(*

short summary
=================
This interface provides assert statements for 32 bit ``DATE``  

.. <legal notes>

legal notes
=================
| SPDX-FileCopyrightText: © 2022 ekvip automation GmbH <info@ekvip.de>
| SPDX-License-Identifier: Apache-2.0
| For details check: Apache-2.0_

.. _Apache-2.0: https://www.apache.org/licenses/LICENSE-2.0

.. </legal notes>

methods
==================

*)

INTERFACE I64BitDateAssertions EXTENDS __SYSTEM.IQueryInterface

(*

short summary
=================
This assertion method checks if the current value is equal to the expected value

.. <legal notes>

legal notes
=================
| SPDX-FileCopyrightText: © 2022 ekvip automation GmbH <info@ekvip.de>
| SPDX-License-Identifier: Apache-2.0
| For details check: Apache-2.0_

.. _Apache-2.0: https://www.apache.org/licenses/LICENSE-2.0

.. </legal notes>

parameters
=================

*)

METHOD valueIsEqualTo
VAR_INPUT
	(* current value to check *)
	currentValue	:LDATE;
	(* expected value to compare *)
	expectedValue	:LDATE;
	(* message if the assertion is false *)
	message			:AssertMessage;
END_VAR
END_METHOD

(*

short summary
=================
This assertion method checks if the current value is greater than the less value

.. <legal notes>

legal notes
=================
| SPDX-FileCopyrightText: © 2022 ekvip automation GmbH <info@ekvip.de>
| SPDX-License-Identifier: Apache-2.0
| For details check: Apache-2.0_

.. _Apache-2.0: https://www.apache.org/licenses/LICENSE-2.0

.. </legal notes>

parameters
=================

*)

METHOD valueIsGreaterThan
VAR_INPUT
	(* current value to check *)
	currentValue	:LDATE;
	(* less than lower limit *)
	lessValue		:LDATE;
	(* message if the assertion is false *)
	message			:AssertMessage;
END_VAR
END_METHOD

(*

short summary
=================
This assertion method checks if the current value is inside a limit

.. attention:: 
	limits are included: ``valueIsInRangeOf(ldate#1970-01-01, ldate#1970-01-01, ldate#1970-01-01)``
	is a true assertion

.. <legal notes>

legal notes
=================
| SPDX-FileCopyrightText: © 2022 ekvip automation GmbH <info@ekvip.de>
| SPDX-License-Identifier: Apache-2.0
| For details check: Apache-2.0_

.. _Apache-2.0: https://www.apache.org/licenses/LICENSE-2.0

.. </legal notes>

parameters
=================

*)

METHOD valueIsInRangeOf
VAR_INPUT
	(* lower limit for the current value *)
	lowerLimit		:LDATE;
	(* current value to check *)
	currentValue	:LDATE;
	(* upper limit for the current value *)
	upperLimit		:LDATE;
	(* message if the assertion is false *)
	message			:AssertMessage;
END_VAR
END_METHOD

(*

short summary
=================
This assertion method checks if the current value is less than the greater value

.. <legal notes>

legal notes
=================
| SPDX-FileCopyrightText: © 2022 ekvip automation GmbH <info@ekvip.de>
| SPDX-License-Identifier: Apache-2.0
| For details check: Apache-2.0_

.. _Apache-2.0: https://www.apache.org/licenses/LICENSE-2.0

.. </legal notes>

parameters
=================

*)

METHOD valueIsLessThan
VAR_INPUT
	(* current value to check *)
	currentValue	:LDATE;
	(* greater than upper limit *)
	greaterValue	:LDATE;
	(* message if the assertion is false *)
	message			:AssertMessage;
END_VAR
END_METHOD

(*

short summary
=================
This assertion method checks if the current value is less than or equal to the maximum value

.. <legal notes>

legal notes
=================
| SPDX-FileCopyrightText: © 2022 ekvip automation GmbH <info@ekvip.de>
| SPDX-License-Identifier: Apache-2.0
| For details check: Apache-2.0_

.. _Apache-2.0: https://www.apache.org/licenses/LICENSE-2.0

.. </legal notes>

parameters
=================

*)

METHOD valueIsMax
VAR_INPUT
	(* current value to check *)
	currentValue	:LDATE;
	(* upper limit for the current value *)
	maximumValue	:LDATE;
	(* message if the assertion is false *)
	message			:AssertMessage;
END_VAR
END_METHOD

(*

short summary
=================
This assertion method checks if the current value is greater than or equal to the minimum value

.. <legal notes>

legal notes
=================
| SPDX-FileCopyrightText: © 2022 ekvip automation GmbH <info@ekvip.de>
| SPDX-License-Identifier: Apache-2.0
| For details check: Apache-2.0_

.. _Apache-2.0: https://www.apache.org/licenses/LICENSE-2.0

.. </legal notes>

parameters
=================

*)

METHOD valueIsMin
VAR_INPUT
	(* current value to check *)
	currentValue	:LDATE;
	(* lower limit for the current value *)
	minimumValue	:LDATE;
	(* message if the assertion is false *)
	message			:AssertMessage;
END_VAR
END_METHOD

(*

short summary
=================
This assertion method checks if the current value is not equal to the unexpected value

.. <legal notes>

legal notes
=================
| SPDX-FileCopyrightText: © 2022 ekvip automation GmbH <info@ekvip.de>
| SPDX-License-Identifier: Apache-2.0
| For details check: Apache-2.0_

.. _Apache-2.0: https://www.apache.org/licenses/LICENSE-2.0

.. </legal notes>

parameters
=================

*)

METHOD valueIsNotEqualTo
VAR_INPUT
	(* current value to check *)
	currentValue	:LDATE;
	(* unexpected value to compare *)
	unexpectedValue	:LDATE;
	(* message if the assertion is false *)
	message			:AssertMessage;
END_VAR
END_METHOD

END_INTERFACE

(* stored: Version 1.1.0.1, ProductVersion 3.1.4026.8
   Itf I64BitDateAssertions: Id {822ae77e-1cf7-43ca-9abe-bb34b6d90df6}
   Method valueIsEqualTo: Id {456ee973-1d8e-4ac2-ad6c-9f70966f6113}
   Method valueIsGreaterThan: Id {3fef51b9-a208-4dfc-b692-d8eba27cf7cb}
   Method valueIsInRangeOf: Id {99df9eba-c040-4381-9125-656f45c0e389}
   Method valueIsLessThan: Id {061657bb-0633-46f9-abf0-f8af16865adf}
   Method valueIsMax: Id {91dda0ea-c081-4280-b2e2-e7800a0d6a32}
   Method valueIsMin: Id {ec67ab4e-e347-4e98-b41f-47034769749b}
   Method valueIsNotEqualTo: Id {e9762fb9-1e84-4d5a-97cb-4874ec475f85} *)
